// TIA Portal V19 export
FUNCTION_BLOCK "MainFB"   // FB10, FBD
TITLE = MainFB
{ S7_Optimized_Access := 'TRUE' }
AUTHOR : Siemens
// Main FB BeltLift
// stored: IsIECCheckEnabled true, MemoryReserve 100, SetENOAutomatically true
   VAR_INPUT
      Initial_Call { ExternalAccessible := 'False'; ExternalVisible := 'False'; ExternalWritable := 'False'} : Bool;   // Initial call of this OB
   END_VAR
   VAR
      instCommon { ExternalAccessible := 'False'; ExternalVisible := 'False'; ExternalWritable := 'False'; S7_SetPoint := 'True'} : "Common";
      instLift1Cmd { ExternalAccessible := 'False'; ExternalVisible := 'False'; ExternalWritable := 'False'; S7_SetPoint := 'True'} : "LiftCmd";
      instLift2Cmd { ExternalAccessible := 'False'; ExternalVisible := 'False'; ExternalWritable := 'False'; S7_SetPoint := 'True'} : "LiftCmd";
      instLiftSim { ExternalAccessible := 'False'; ExternalVisible := 'False'; ExternalWritable := 'False'; S7_SetPoint := 'True'} : "LiftSim";
   END_VAR
BEGIN

REGION Network 1: common
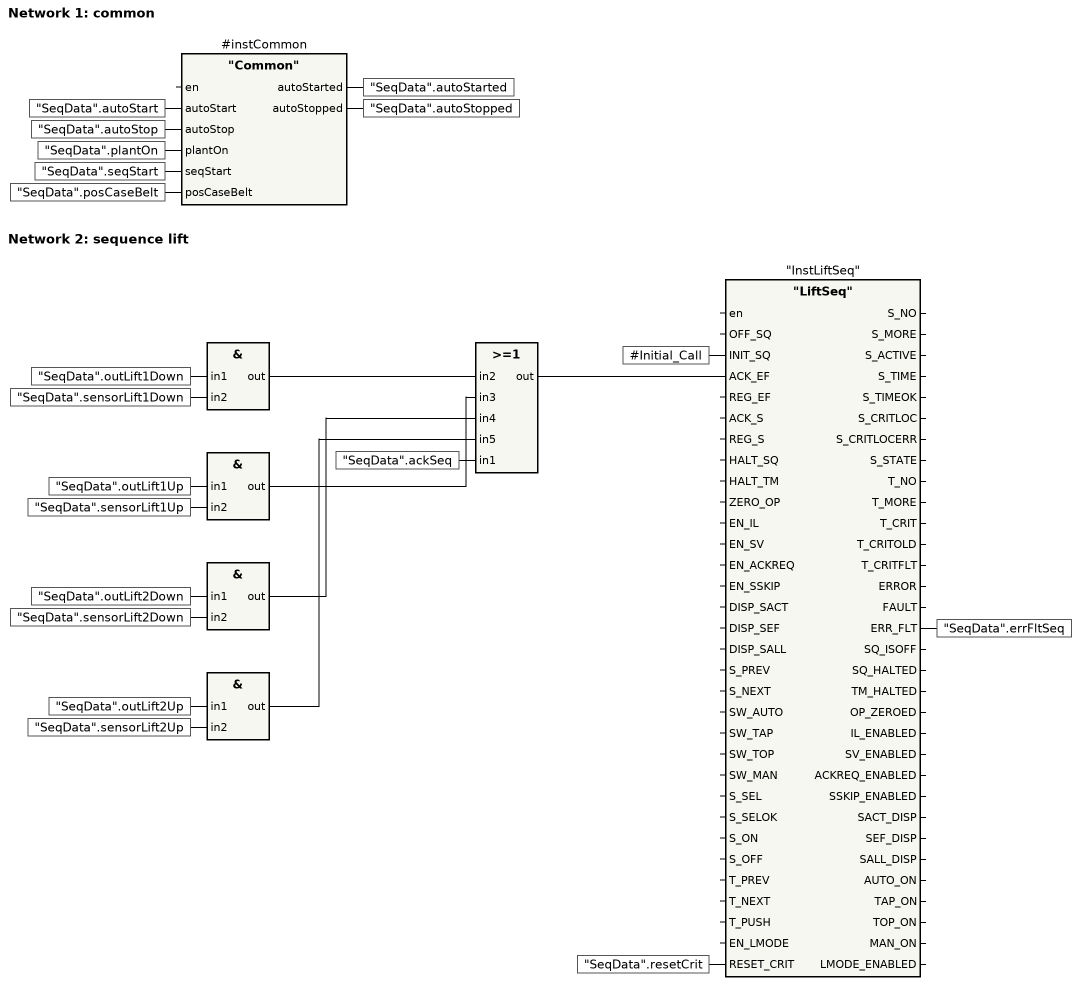
   #instCommon(autoStart := "SeqData".autoStart,   // "Common"
               autoStop := "SeqData".autoStop,
               plantOn := "SeqData".plantOn,
               seqStart := "SeqData".seqStart,
               posCaseBelt := "SeqData".posCaseBelt,
               autoStarted => "SeqData".autoStarted,
               autoStopped => "SeqData".autoStopped);
END_REGION

REGION Network 2: sequence lift
   "InstLiftSeq"(INIT_SQ := #Initial_Call,   // "LiftSeq"
                 ACK_EF := ("SeqData".outLift1Down AND "SeqData".sensorLift1Down) OR ("SeqData".outLift1Up AND "SeqData".sensorLift1Up) OR ("SeqData".outLift2Down AND "SeqData".sensorLift2Down) OR ("SeqData".outLift2Up AND "SeqData".sensorLift2Up) OR "SeqData".ackSeq,
                 RESET_CRIT := "SeqData".resetCrit,
                 ERR_FLT => "SeqData".errFltSeq);
END_REGION

REGION Network 3: Lift 1
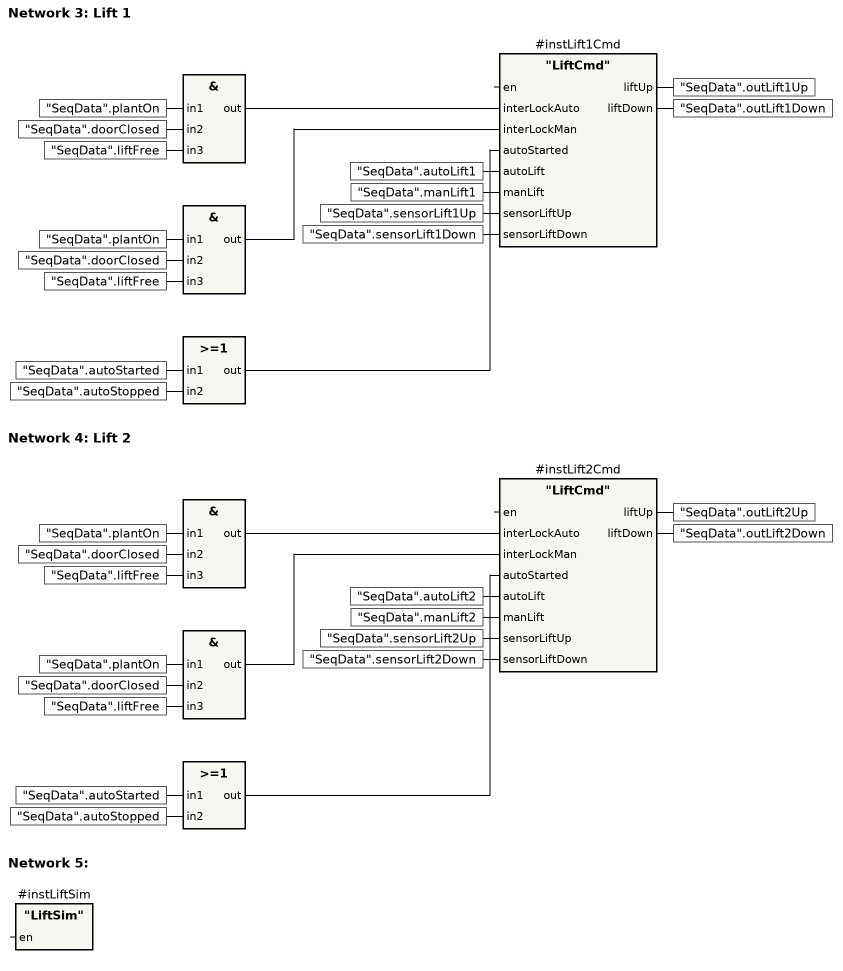
   #instLift1Cmd(interLockAuto := "SeqData".plantOn AND "SeqData".doorClosed AND "SeqData".liftFree,   // "LiftCmd"
                 interLockMan := "SeqData".plantOn AND "SeqData".doorClosed AND "SeqData".liftFree,
                 autoStarted := "SeqData".autoStarted OR "SeqData".autoStopped,
                 autoLift := "SeqData".autoLift1,
                 manLift := "SeqData".manLift1,
                 sensorLiftUp := "SeqData".sensorLift1Up,
                 sensorLiftDown := "SeqData".sensorLift1Down,
                 liftUp => "SeqData".outLift1Up,
                 liftDown => "SeqData".outLift1Down);
END_REGION

REGION Network 4: Lift 2
   #instLift2Cmd(interLockAuto := "SeqData".plantOn AND "SeqData".doorClosed AND "SeqData".liftFree,   // "LiftCmd"
                 interLockMan := "SeqData".plantOn AND "SeqData".doorClosed AND "SeqData".liftFree,
                 autoStarted := "SeqData".autoStarted OR "SeqData".autoStopped,
                 autoLift := "SeqData".autoLift2,
                 manLift := "SeqData".manLift2,
                 sensorLiftUp := "SeqData".sensorLift2Up,
                 sensorLiftDown := "SeqData".sensorLift2Down,
                 liftUp => "SeqData".outLift2Up,
                 liftDown => "SeqData".outLift2Down);
END_REGION

REGION Network 5
   #instLiftSim();   // "LiftSim"
END_REGION
END_FUNCTION_BLOCK
